(* CODESYS project lorapayloaddecoder.library
   Company: PXL-Tech
   Title: Lora Payload Decoder
   Placeholder: Lora Payload Decoder
   Version: 1.0

Project tree, tasks and I/O mapping:
  libraries: Tc2_Standard, * (Beckhoff Automation GmbH); Tc2_System, * (Beckhoff Automation GmbH); Tc2_Utilities, * (Beckhoff Automation GmbH); Tc3_Module, * (Beckhoff Automation GmbH)
  DUTs/
    data type Alarm
    data type Alive
    data type Analog
    data type DailyReport
    data type DigIn1Msg
    data type DigIn2Msg
    data type GenSens
    data type GenSensGravMsg
    data type Indoor
    data type OneWireT
    data type Reboot
    data type Rot
    data type Running
    data type Shock
    data type Tracking
    data type Vibrate
  GVLs/
  POUs/
    function block FB_PayloadDecoder [ST]
    program MAIN [ST]
  Version/
    global variables Global_Version
  VISUs/
*)

// DUTs/Alarm
TYPE Alarm :
STRUCT
	GravRotAl		:BOOL;	// Gravity Rotation Detected
	MagRot			:BOOL;	// Magnetic Rotation Detected
	MotAlarm		:BOOL;	// Motion Alarm Detected
	GeoFenceAl		:BOOL;	// GeoFence Violation Detected
	VibrAl			:BOOL;	// Vibration Alarm Detected
	ShockAl			:BOOL;	// Shock Alarm (future use)
	DigIn1Al		:BOOL;	// Digin1 Alarm Detected
	DigIn2Al		:BOOL;	// Digin2 Alarm Detected
	Temp			:REAL;	// Temperature in 0,01 Celcius
	Hum				:BYTE;	// Relative Humidity in %
	BaromBar		:REAL;	// Air Pressure in Mbar
END_STRUCT
END_TYPE

// DUTs/Alive
TYPE Alive :
STRUCT
	Battery			:BYTE;					// 0..255 == 0%..100%
	DigIn1			:BOOL;					// DigIn1 State
	DigIn2			:BOOL;					// DigIn2 State
	Spare1			:BOOL;					// Spare
	Spare2			:BOOL;					// Spare
	Spare3			:BOOL;					// Spare
	Spare4			:BOOL;					// Spare
	Spare5			:BOOL;					// Spare
	PowerOut	    :BOOL;					// +5V Output State
	CmdAck			:BYTE;					// Sequence number of last received Command
	GPSFixAge		:BYTE;					// bit 0..7 = Age of last GPS Fix in Minutes MsgIDsee above),
	SatCnt_HiLL		:BYTE;					// bit 0..4 = SatInFix, bit5 Latitude 24bit 6,7 = Longitude 24,25
	Lat				:REAL;
	Lon				:REAL;
END_STRUCT
END_TYPE

// DUTs/Analog
TYPE Analog :
STRUCT
	VBat				:INT;	// Battery voltage in mV
	AnalogIn1			:INT;	// AnalogIn 1 in mV
	AnalogIn2			:INT;	// AnalogIn 2 in mV
	AnalogIn3			:INT;	// Distance measurement for Sonar
	Analogin4			:INT;	// future use
END_STRUCT
END_TYPE

// DUTs/DailyReport
TYPE DailyReport :
STRUCT
	Status			:BYTE;	// Content Depends on Message ID for future use
	MinTemp			:REAL;	// Minimum Temperature DgrC -27..+100 DgrC since last DailyRep Message
	MaxTemp			:REAL;	// Maximum Temperature DgrC -27..+100 DgrC sincelast DailyRep Message
	MinHum			:BYTE;	// Minimum Humidity since last DailyRep Message
	MaxHum			:BYTE;	// Maximum Humidity since last DailyRep Message
	MaxBaro			:BYTE;	// Maximum Barosince last DailyRep Message
	MinBaro			:BYTE;	// Minimum Barosince last DailyRep Message
	RunHrs			:WORD;	// Running Hours (in hours)
	KM				:WORD;	// Distance traveled in KM
END_STRUCT
END_TYPE

// DUTs/DigIn1Msg
TYPE DigIn1Msg :
STRUCT
	Mode			:BYTE;	// Current Digin1 Mode
	RepMode			:BYTE;	// Current Digin Report Moded
	Counter			:DWORD;	// Digin1 Counterd
	RunTimer		:DWORD;	// Digin1 RunTimer (seconds)
	State			:BYTE;	// State of Digin1
END_STRUCT
END_TYPE

// DUTs/DigIn2Msg
TYPE DigIn2Msg :
STRUCT
	Mode			:BYTE;	// Current Digin2 Mode
	RepMode			:BYTE;	// Current Digin Report Moded
	Counter			:DWORD;	// Digin2 Counterd
	RunTimer		:DWORD;	// Digin2 RunTimer (seconds)
	State			:BYTE;	// State of Digin2
END_STRUCT
END_TYPE

// DUTs/GenSens
TYPE GenSens :
STRUCT
	Status     			:BYTE;      // Content Depends on Message ID == for future use
	BaromBar			:REAL;      // Air Pressure in mBar
	Temp   				:REAL;     	// in 0,01 degC
	Humidity   			:BYTE;      // Relative Humidity in %
	LevelX     			:SINT;      // Inverse Sinus of Spirit Level in Deg X-Direction -128 = -90 Degr .. +127 = +90 Degr
	LevelY     			:SINT;      // Inverse Sinus of Spirit Level in Deg Y-Direction -128 = -90 Degr .. +127 = +90 Degr
	LevelZ     			:SINT;      // Inverse Sinus of Spirit Level in Deg Z-Direction -128 = -90 Degr .. +127 = +90 Degr
	VibAmp     			:USINT;     // Amplitude of Vibration Detected == Future
	VibFreq    			:USINT;     // Approx. Frequency of Vibration Detected in Hz == Future
END_STRUCT
END_TYPE

// DUTs/GenSensGravMsg
TYPE GenSensGravMsg :
STRUCT
	Status     			:BYTE;      // Content Depends on Message ID == for future use
	BaromBar			:REAL;      // Air Pressure in mBar
	Temp				:REAL;     	// in 0,01 degC
	Humidity   			:BYTE;      // Relative Humidity in %
	GravX     			:SINT;      // Accelerometer X
	GravY     			:SINT;      // Accelerometer Y
	GravZ     			:SINT;      // Accelerometer Z
	VibAmp     			:USINT;     // Amplitude of Vibration Detected == Future
	VibFreq    			:USINT;     // Approx. Frequency of Vibration Detected in Hz = Future
END_STRUCT
END_TYPE

// DUTs/Indoor
TYPE Indoor :
STRUCT
	Start				:BOOL;	// Start Message
	Moving	 			:BOOL;	// Object Moving
	Stop				:BOOL;	// Object Stopped
	Vibr				:BOOL;	// Vibration Detected
	BeaconID1			:WORD;	// ID of beacon 1(16 bits of DEVEUI)
	RSSI1				:SINT;	// RSSI of Beacon1
	BeaconID2			:WORD;	// ID of beacon 2(16 bits of DEVEUI)
	RSSI2				:SINT;	// RSSI of Beacon2
	BeaconID3			:WORD;	// ID of beacon 3(16 bits of DEVEUI)
	RSSI3				:SINT;	// RSSI of Beacon3
	RFU1				:BYTE;
END_STRUCT
END_TYPE

// DUTs/OneWireT
TYPE OneWireT :
STRUCT
	NumOfSensors		:BYTE;		// Number of 1Wire sensors currently connected
	Sens1ID				:BYTE;		// Sensor ShortID
	Sens1Temp			:REAL;		// in 0,1 degC
	Sens2ID				:BYTE;		// Sensor ShortID
	Sens2Temp			:REAL;		// in 0,1 degC
	Sens3ID				:BYTE;		// Sensor ShortID
	Sens3Temp			:REAL;		// in 0,1 degC
	Sens4ID				:BYTE;		// Sensor ShortID
	Sens4Temp			:REAL;		// in 0,1 degC
	Sens5ID				:BYTE;		// Sensor ShortID
	Sens5Temp			:REAL;		// in 0,1 degC
END_STRUCT
END_TYPE

// DUTs/Reboot
TYPE Reboot :
STRUCT
	RebootReason		:BYTE;		// For internal use
	Profile				:USINT;		// For internal use
	CmdAck				:USINT;		// Last received Command
	OneM2MID			:DWORD;		// 1M2M Serial number
	SrcID				:BYTE;		// Rebootreason source file ID incl.reboot reason
	LineNR				:WORD;		// Reboot reason line number 
	Version				:BYTE;		// Firmware Version bit 0..3 Low  4..7 High
END_STRUCT
END_TYPE

// DUTs/Rot
TYPE Rot :
STRUCT
	GravRotAl		:BOOL;	// Gravity Rotation Detected
	MagRot			:BOOL;	// Mag Rotation Detected
	GravX			:SINT;	// Gravity in X-Direction 64 ~~ 1G 
	GravY			:SINT;	// Gravity in Y-Direction 64 ~~ 1G 
	GravZ			:SINT;	// Gravity in Z-Direction 64 ~~ 1G 
	MagX			:SINT;	// Magnetic Field in X-direction 10 uTesla
	MagY			:SINT;	// Magnetic Field in Y-direction 10 uTesla
	MagZ			:SINT;	// Magnetic Field in Z-direction 10 uTesla
END_STRUCT
END_TYPE

// DUTs/Running
TYPE Running :
STRUCT
	MaxFreq1	:BYTE;
	MaxAmpl1	:BYTE;
	MaxFreq2	:BYTE;
	MaxAmpl2	:BYTE;
	MaxFreq3	:BYTE;
	MaxAmpl3	:BYTE;
END_STRUCT
END_TYPE

// DUTs/Shock
TYPE Shock :
STRUCT
	Impact				:BYTE;	// The average of the FFT values over X+Y+Z < 30Hz(experimental)
	Shock				:WORD;	// Maximum Measured Acceleration in combined directionXYZ
	MaxDx				:WORD;	// Max Acceleration in X-direction 
	MaxDy				:WORD;	// Max Acceleration in Y-direction
	MaxDz				:WORD;	// Max Acceleration in Z-direction
	Range				:BYTE;	// Accelerometer Range 0 = 2G; 1= 4G; 2 = 8G; 3 = 16G
	NumOfShocks			:BYTE;	// Number of Shocks
END_STRUCT
END_TYPE

// DUTs/Tracking
TYPE Tracking :
STRUCT
	Start				:BOOL;// Start Message
	Moving				:BOOL;// Object Moving
	Stop				:BOOL;// Object Stopped
	Vibr				:BOOL;// Vibration Detected
	Temp				:REAL;// Temperature in 0,01 degC
	GPSFixAge			:BYTE;// bit 0..7 = Age of last GPS Fix in Minutes,
	SatCnt_HiLL			:BYTE;// bit 0..4 = SatInFix, bit5 Latitude 25 bit 6,7 = Longitude 25,26
	Lat					:REAL;
	Lon					:REAL;
END_STRUCT
END_TYPE

// DUTs/Vibrate
TYPE Vibrate :
STRUCT
	MaxdX				:BYTE;	// Maximum deviation in AccelerometerX
	MaxdY				:BYTE;	// Maximum deviation in AccelerometerY
	MaxdZ				:BYTE;	// Maximum deviation in AccelerometerZ
	Max1Freq			:UINT;	// Frequency with highest amplitude
	Max1Ampl			:BYTE;	// Amplitude of Frequency with highest Amplitude
	Max2Freq			:UINT;	// Frequency with second highest amplitude
	Max2Ampl			:BYTE;	// Amplitude of Frequency with second highest Amplitude
	Max3Freq			:UINT;	// Frequency with third highest amplitude
	Max3Ampl			:BYTE;	// Amplitude of Frequency with third highest Amplitude
	vAgcVibr			:BYTE;	// Gain Value Vibration Detection 0x00=2G, 0x01=4G,0x02=8G, 0x03=16G
END_STRUCT
END_TYPE

// Version/Global_Version
{attribute 'TcGenerated'}
// This function has been automatically generated from the project information.
VAR_GLOBAL CONSTANT
	{attribute 'const_non_replaced'}
	{attribute 'linkalways'}
	stLibVersion_Lora_Payload_Decoder : ST_LibVersion := (iMajor := 1, iMinor := 0, iBuild := 0, iRevision := 0, sVersion := '1.0');
END_VAR

// POUs/FB_PayloadDecoder
FUNCTION_BLOCK FB_PayloadDecoder
VAR_INPUT
	dataString :STRING(32);
END_VAR
VAR_OUTPUT
	MsgID      		:	BYTE;
	
	Alive 			:	Alive;			//0x00
	Tracking		:	Tracking;		//0x01
	GenSens			:	GenSens;		//0x02
	Rot				:	Rot;			//0x03
	Alarm			:	Alarm;			//0x04
	OneWireT		:	OneWireT;		//0x06
	Running			:	Running;		//0x07
	Vibrate			:	Vibrate;		//0x08
	Analog			:	Analog;			//0x09
	GenSensGravMsg	:	GenSensGravMsg;	//0x0A
	DailyReport		:	DailyReport;	//0x0B
	DigIn1Msg		:	DigIn1Msg;		//0x0C
	DigIn2Msg		:	DigIn2Msg;		//0x0D
	Indoor			:	Indoor;			//0x81
	Shock			:	Shock;			//0x82
	Reboot			:	Reboot;			//0x0E
	
	
END_VAR
VAR
	dataBuf       :ARRAY[1..16] OF BYTE;
	
	Adress: POINTER TO WORD;
END_VAR

HEXSTR_TO_DATA(dataString, ADR(dataBuf), SIZEOF(dataBuf));

MsgID := dataBuf[1];
CASE MsgID OF
	16#00:
		Alive.Battery := dataBuf[2];
		Alive.DigIn1 := USINT_TO_BOOL(dataBuf[3] AND 1);
		Alive.DigIn2 := USINT_TO_BOOL(SHR(dataBuf[3], 1) AND 1);
		Alive.Spare1 := USINT_TO_BOOL(SHR(dataBuf[3], 2) AND 1);
		Alive.Spare2 := USINT_TO_BOOL(SHR(dataBuf[3], 3) AND 1);
		Alive.Spare3 := USINT_TO_BOOL(SHR(dataBuf[3], 4) AND 1);
		Alive.Spare4 := USINT_TO_BOOL(SHR(dataBuf[3], 5) AND 1);
		Alive.Spare5 := USINT_TO_BOOL(SHR(dataBuf[3], 6) AND 1);
		Alive.PowerOut := USINT_TO_BOOL(SHR(dataBuf[3], 7) AND 1);
		Alive.CmdAck := dataBuf[4];
		Alive.GPSFixAge := dataBuf[5];
		Alive.SatCnt_HiLL := dataBuf[6];
		Alive.Lat := DWORD_TO_REAL(SHL(dataBuf[7], 16) OR SHL(dataBuf[8], 8) OR dataBuf[9]) / 100000;
		Alive.Lon := DWORD_TO_REAL(SHL(dataBuf[10], 16) OR SHL(dataBuf[11], 8) OR dataBuf[12]) / 100000;
	16#01:
		Tracking.Start := USINT_TO_BOOL(dataBuf[2] AND 1);
		Tracking.Moving := USINT_TO_BOOL(SHR(dataBuf[2], 1) AND 1);
		Tracking.Stop := USINT_TO_BOOL(SHR(dataBuf[2], 2) AND 1);
		Tracking.Vibr := USINT_TO_BOOL(SHR(dataBuf[2], 3) AND 1);
		Tracking.Temp := UINT_TO_REAL(SHL(dataBuf[3], 8) OR dataBuf[4]) / 100;
		Tracking.GPSFixAge := dataBuf[5];
		Tracking.SatCnt_HiLL := dataBuf[6];
		Tracking.Lat := DWORD_TO_REAL(SHL(dataBuf[7], 16) OR SHL(dataBuf[8], 8) OR dataBuf[9]) / 100000;
		Tracking.Lon := DWORD_TO_REAL(SHL(dataBuf[10], 16) OR SHL(dataBuf[11], 8) OR dataBuf[12]) / 100000;
	16#02:
		GenSens.Status := dataBuf[2];
		GenSens.BaromBar := (WORD_TO_REAL(SHL(dataBuf[3], 8) OR dataBuf[4]) + 100000) / 100;
		GenSens.Temp := WORD_TO_REAL(SHL(dataBuf[5], 8) OR dataBuf[6]) / 100;
		GenSens.Humidity := dataBuf[7];
		GenSens.LevelX := BYTE_TO_SINT(dataBuf[8]);
		GenSens.LevelY := BYTE_TO_SINT(dataBuf[9]);
		GenSens.LevelZ := BYTE_TO_SINT(dataBuf[10]);
		GenSens.VibAmp := dataBuf[11];
		GenSens.VibFreq := dataBuf[12];
	16#03:
		Rot.GravRotAl := USINT_TO_BOOL(dataBuf[2] AND 1);
		Rot.MagRot := USINT_TO_BOOL(SHR(dataBuf[2], 1) AND 1);
		Rot.GravX := DataBuf[3];
		Rot.GravY := DataBuf[4];
		Rot.GravZ := DataBuf[5];
		Rot.MagX := DataBuf[6];
		Rot.MagY := DataBuf[7];
		Rot.MagZ := DataBuf[8];
	16#04:
		Alarm.GravRotAl := USINT_TO_BOOL(dataBuf[2] AND 1);
		Alarm.MagRot := USINT_TO_BOOL(SHR(dataBuf[2], 1) AND 1);
		Alarm.MotAlarm := USINT_TO_BOOL(SHR(dataBuf[2], 2) AND 1);
		Alarm.GeoFenceAl := USINT_TO_BOOL(SHR(dataBuf[2], 3) AND 1);
		Alarm.VibrAl := USINT_TO_BOOL(SHR(dataBuf[2], 4) AND 1);
		Alarm.ShockAl := USINT_TO_BOOL(SHR(dataBuf[2], 5) AND 1);
		Alarm.DigIn1Al := USINT_TO_BOOL(SHR(dataBuf[2], 6) AND 1);
		Alarm.DigIn2Al := USINT_TO_BOOL(SHR(dataBuf[2], 7) AND 1);
		Alarm.Temp := WORD_TO_REAL(SHL(dataBuf[5], 8) OR dataBuf[6]) / 100;
		Alarm.Hum := DataBuf[7];
		Alarm.BaromBar := (WORD_TO_REAL(SHL(dataBuf[8], 8) OR dataBuf[9]) + 100000) / 100;
	16#06:
		OneWireT.NumOfSensors := DataBuf[2];
		IF OneWireT.NumOfSensors > 0 THEN
			OneWireT.Sens1ID := SHR(dataBuf[3], 4);
			OneWireT.Sens1Temp := (WORD_TO_REAL(SHL(dataBuf[3] AND 16#0F, 8) OR dataBuf[4]) - 550) / 10;
		END_IF
		IF OneWireT.NumOfSensors > 1 THEN
			OneWireT.Sens2ID := SHR(dataBuf[3], 4);
			OneWireT.Sens2Temp := (WORD_TO_REAL(SHL(dataBuf[3] AND 16#0F, 8) OR dataBuf[4]) - 550) / 10;
		END_IF
		IF OneWireT.NumOfSensors > 2 THEN
			OneWireT.Sens3ID := SHR(dataBuf[5], 4);
			OneWireT.Sens3Temp := (WORD_TO_REAL(SHL(dataBuf[5] AND 16#0F, 8) OR dataBuf[6]) - 550) / 10;
		END_IF
		IF OneWireT.NumOfSensors > 3 THEN
			OneWireT.Sens4ID := SHR(dataBuf[7], 4);
			OneWireT.Sens4Temp := (WORD_TO_REAL(SHL(dataBuf[7] AND 16#0F, 8) OR dataBuf[8]) - 550) / 10;
		END_IF
		IF OneWireT.NumOfSensors > 4 THEN
			OneWireT.Sens5ID := SHR(dataBuf[9], 4);
			OneWireT.Sens5Temp := (WORD_TO_REAL(SHL(dataBuf[9] AND 16#0F, 8) OR dataBuf[10]) - 550) / 10;
		END_IF
	16#07:
		Running.MaxFreq1 := dataBuf[6];
		Running.MaxAmpl1 := dataBuf[7];
		Running.MaxFreq2 := dataBuf[8];
		Running.MaxAmpl2 := dataBuf[9];
		Running.MaxFreq3 := dataBuf[10];
		Running.MaxAmpl3 := dataBuf[11];
	16#08:
		Vibrate.MaxdX := dataBuf[2];
		Vibrate.MaxdY := dataBuf[3];
		Vibrate.MaxdZ := dataBuf[4];
		Vibrate.Max1Freq := BYTE_TO_UINT(dataBuf[5]) * 630 / 53;
		Vibrate.Max1Ampl := dataBuf[6];
		Vibrate.Max2Freq := BYTE_TO_UINT(dataBuf[7]) * 630 / 53;
		Vibrate.Max2Ampl := dataBuf[8];
		Vibrate.Max3Freq := BYTE_TO_UINT(dataBuf[9]) * 630 / 53;
		Vibrate.Max3Ampl := dataBuf[10];
		Vibrate.vAgcVibr := dataBuf[11];	
	16#09:
		Analog.VBat := 	SHL(dataBuf[2], 8) OR dataBuf[3];
		Analog.AnalogIn1 := SHL(dataBuf[4], 8) OR dataBuf[5];
		Analog.AnalogIn2 := SHL(dataBuf[6], 8) OR dataBuf[7];
		Analog.AnalogIn3 := SHL(dataBuf[8], 8) OR dataBuf[9];
		Analog.AnalogIn4 := SHL(dataBuf[10], 8) OR dataBuf[11];
	16#0A:
		GenSensGravMsg.Status := dataBuf[2];
		GenSensGravMsg.BaromBar := (WORD_TO_REAL(SHL(dataBuf[3], 8) OR dataBuf[4]) + 100000) / 100;
		GenSensGravMsg.Temp := WORD_TO_REAL(SHL(dataBuf[5], 8) OR dataBuf[6]) / 100;
		GenSensGravMsg.Humidity := dataBuf[7];
		GenSensGravMsg.GravX := BYTE_TO_SINT(dataBuf[8]);
		GenSensGravMsg.GravY := BYTE_TO_SINT(dataBuf[9]);
		GenSensGravMsg.GravZ := BYTE_TO_SINT(dataBuf[10]);
		GenSensGravMsg.VibAmp := dataBuf[11];
		GenSensGravMsg.VibFreq := dataBuf[12];
	16#0B:
		DailyReport.Status := dataBuf[2];
		DailyReport.MinTemp := BYTE_TO_REAL(dataBuf[3]) / 100;
		DailyReport.MaxTemp := BYTE_TO_REAL(dataBuf[4]) / 100;
		DailyReport.MinHum := dataBuf[5];
		DailyReport.MaxHum := dataBuf[6];
		DailyReport.MaxBaro := dataBuf[7];
		DailyReport.MinBaro := dataBuf[8];
		DailyReport.RunHrs := SHL(dataBuf[9], 8) OR dataBuf[10];
		DailyReport.KM := SHL(dataBuf[11], 8) OR dataBuf[12];
	16#0C:
		DigIn1Msg.Mode := dataBuf[2];
		DigIn1Msg.RepMode := dataBuf[3];
		DigIn1Msg.Counter := SHL(dataBuf[4], 24) OR SHL(dataBuf[5], 16) OR SHL(dataBuf[6], 8) OR dataBuf[7];
		DigIn1Msg.RunTimer := SHL(dataBuf[8], 24) OR SHL(dataBuf[9], 16) OR SHL(dataBuf[10], 8) OR dataBuf[11];
		DigIn1Msg.State := dataBuf[12];
	16#0D:
		DigIn2Msg.Mode := dataBuf[2];
		DigIn2Msg.RepMode := dataBuf[3];
		DigIn2Msg.Counter := SHL(dataBuf[4], 24) OR SHL(dataBuf[5], 16) OR SHL(dataBuf[6], 8) OR dataBuf[7];
		DigIn2Msg.RunTimer := SHL(dataBuf[8], 24) OR SHL(dataBuf[9], 16) OR SHL(dataBuf[10], 8) OR dataBuf[11];
		DigIn2Msg.State := dataBuf[12];
	16#81:
		Indoor.Start := USINT_TO_BOOL(dataBuf[2] AND 1);
		Indoor.Moving := USINT_TO_BOOL(SHR(dataBuf[2], 1) AND 1);
		Indoor.Stop := USINT_TO_BOOL(SHR(dataBuf[2], 2) AND 1);
		Indoor.Vibr := USINT_TO_BOOL(SHR(dataBuf[2], 3) AND 1);
		Indoor.BeaconID1 := SHL(dataBuf[3], 8) OR dataBuf[4];
		Indoor.RSSI1 := BYTE_TO_SINT(dataBuf[5]);
		Indoor.BeaconID2 := SHL(dataBuf[6], 8) OR dataBuf[7];
		Indoor.RSSI2 := BYTE_TO_SINT(dataBuf[8]);
		Indoor.BeaconID3 := SHL(dataBuf[9], 8) OR dataBuf[10];
		Indoor.RSSI3 := BYTE_TO_SINT(dataBuf[11]);
		Indoor.RFU1 := dataBuf[12];
	16#82:
		Shock.Impact := dataBuf[2];
		Shock.Shock := SHL(dataBuf[3], 8) OR dataBuf[4];
		Shock.MaxDx := SHL(dataBuf[5], 8) OR dataBuf[6];
		Shock.MaxDy := SHL(dataBuf[7], 8) OR dataBuf[8];
		Shock.MaxDz := SHL(dataBuf[9], 8) OR dataBuf[10];
		Shock.Range := dataBuf[11];
		Shock.NumOfShocks := dataBuf[12];			
	16#0E:
		Reboot.RebootReason := dataBuf[2];
		Reboot.Profile := dataBuf[3];
		Reboot.CmdAck := dataBuf[4];
		Reboot.OneM2MID := SHL(dataBuf[5], 24) OR SHL(dataBuf[6], 16) OR SHL(dataBuf[7], 8) OR dataBuf[8];
		Reboot.SrcID := dataBuf[9];
		Reboot.LineNR := SHL(dataBuf[10], 8) OR dataBuf[11];
		Reboot.Version := dataBuf[12];
END_CASE

END_FUNCTION_BLOCK

// POUs/MAIN
PROGRAM MAIN
VAR
	fb_Decoder : FB_PayloadDecoder;
	dataStr :STRING(32) := '810102030405060708090A0B0C0D0E0F'; // example : 020006250a3b2bc60073000000000000 or 010102030405060708090A0B0C0D0E0F
	temperature : REAL;
END_VAR

fb_Decoder(dataString := dataStr);

END_PROGRAM
